// TIA Portal V17 export
// export: Created 2025-08-05T09:36:00.1761583Z, ExportSetting WithDefaults, DisplayName Totally Integrated Automation Portal, DisplayVersion V17, DisplayName TIA Portal Openness, DisplayVersion V17, DisplayName TIA Portal Version Control Interface, DisplayVersion V17, DisplayName SINAMICS Startdrive Advanced, DisplayVersion V17, DisplayName SINAMICS Startdrive G130, G150, S120, S150, SINAMICS MV, S210, DisplayVersion V17, DisplayName SINAMICS Startdrive G110M, G120, G120C, G120D, G120P, G115D, DisplayVersion V17, DisplayName STEP 7 Professional, DisplayVersion V17, DisplayName STEP 7 Safety, DisplayVersion V17, DisplayName WinCC Advanced, DisplayVersion V17
TYPE "typeHmiScreen"
TITLE = Manual HMI operating screens / HMI Handbedienbilder
// HMI manual operation screens [V 01.00 | Kernel_V2] / HMI Handbedienbilder [V 01.00 | Kernel_V2]
// stored: IsFailsafeCompliant false
   STRUCT
      setup : Struct   // Handbedienbild Einrichten / Manual operating screen 'Setup'
         activ : Bool;   // Aktiv / Active
      END_STRUCT;
      powerup : Struct   // Handbedienbild Einschaltbedingung / Manual operating screen 'Switch-on condition'
         activ : Bool;   // Aktiv / Active
      END_STRUCT;
      unit : Struct   // Handbedienbild Einheiten / Manual operating screen 'Units'
         activ : Bool;   // Aktiv / Active
      END_STRUCT;
      nutrunner : Struct   // Handbedienbild Schrauber / Manual operating screen 'Nut runner'
         activ : Bool;   // Aktiv / Active
      END_STRUCT;
      nutrunnerGroup : Struct   // Handbedienbild Schraubergruppen / Manual operating screen 'Nut runner groups'
         activ : Bool;   // Aktiv / Active
      END_STRUCT;
      cycletype : Struct   // Handbedienbild Taktarten / Manual operating screen 'Cycle types'
         activ : Bool;   // Aktiv / Active
      END_STRUCT;
      userDefine : Struct   // Handbedienbild Anwender / Manual operating screen 'User'
         activ : Bool;   // Aktiv / Active
      END_STRUCT;
   END_STRUCT;
END_TYPE
